// TIA Portal V19 export
DATA_BLOCK "DB_ExportFlatCtrlRobot2"   // DB73
{ S7_Optimized_Access := 'TRUE' }
// stored: AutoNumber false, IsOnlyStoredInLoadMemory true, MemoryReserve 100
   VAR RETAIN
      FlatnessRecords { S7_SetPoint := 'True'} : Array[0..200] of "stFlatnessCtrlRecord";
   END_VAR
BEGIN
   FlatnessRecords[1].dtlDataTime := DTL#2025-07-23-18:25:23.687016057;
   FlatnessRecords[1].xFlatnessResult := TRUE;
   FlatnessRecords[1].uiStrokePositionDiskA := 239;
   FlatnessRecords[1].uiStrokePositionDiskB := 236;
   FlatnessRecords[1].uiStrokePositionDiskC := 237;
END_DATA_BLOCK
